IF NOT bGetProgramStateBusy AND intGetProgramStateStep > 0 THEN
	intGetProgramStateStep := 0;
	bRouterBusy := FALSE;
	THIS^.M_LogWarning('M_GetProgramState ended prematurely!');
END_IF
bGetProgramStateBusy := FALSE;

IF NOT bLoadProgramBusy AND intLoadProgramStep > 0 THEN
	intLoadProgramStep := 0;
	bRouterBusy := FALSE;
	THIS^.M_LogWarning('M_LoadProgram ended prematurely!');
END_IF
bLoadProgramBusy := FALSE;

IF NOT bPauseProgramBusy AND intPauseProgramStep > 0 THEN
	intPauseProgramStep := 0;
	bRouterBusy := FALSE;
	THIS^.M_LogWarning('M_PauseProgram ended prematurely!');
END_IF
bPauseProgramBusy := FALSE;

IF NOT bStartProgramBusy AND intStartProgramStep > 0 THEN
	intStartProgramStep := 0;
	bRouterBusy := FALSE;
	THIS^.M_LogWarning('M_StartProgram ended prematurely!');
END_IF
bStartProgramBusy := FALSE;

IF NOT bStopProgramBusy AND intStopProgramStep > 0 THEN
	intStopProgramStep := 0;
	bRouterBusy := FALSE;
	THIS^.M_LogWarning('M_StopProgram ended prematurely!');
END_IF
bStopProgramBusy := FALSE;

IF NOT bResetBusy AND intResetStep > 0 THEN
	intResetStep := 0;
	bRouterBusy := FALSE;
	THIS^.M_LogWarning('M_ResetBusy ended prematurely!');
END_IF
bResetBusy := FALSE;

IF NOT bAbortBusy AND intAbortStep > 0 THEN
	intAbortStep := 0;
	bRouterBusy := FALSE;
	THIS^.M_LogWarning('M_Abort ended prematurely!');
END_IF
bAbortBusy := FALSE;

IF NOT bRouterHelperBusy AND intRouterHelperStep > 0 THEN
	intRouterHelperStep := 0;
	bRouterBusy := FALSE;
	THIS^.M_LogWarning('M_RouterHelper ended prematurely!');
END_IF
bRouterHelperBusy := FALSE;
END_ACTION

(* This method is a template for any methods that use the API. *)
METHOD M_CommandTemplate : BOOL
VAR CONSTANT
	_strCOMMAND_NAME : T_MaxString	:= 'CommandTemplate'; // Name of the API method
	_timeCOMMAND_TIMEOUT : TIME		:= T#30S; // Max time to receive API response
	_strSTART_MSG : T_MaxString		:= 'Routing command...'; // Prints when method starts
	_strEND_MSG : T_MaxString		:= 'Command complete.'; // Prints when method finishes
	_udintERROR_ID : UDINT			:= E_ApiDeviceError.CommandFault; // Error ID to set if command fails
	_strERROR_MSG : T_MaxString		:= 'Command failed!'; // Error message to set if command fails
END_VAR
VAR_INST
	_inst_arrParams: T_ApiParameterList; // Parameters array
	_inst_arrOutputs: T_ApiParameterList; // Outputs array
	_inst_strRet: T_ApiParamValue; // Return string from the router
	_inst_intStep: INT; // Current method step
	_inst_fbParams: FB_ApiParamBuilder; // Parameter builder FB
END_VAR
VAR
	_bComplete: BOOL; // True if the routing finishes
	_intRet: INT; // Return string converted to an integer
	_bResult : BOOL; // Output of the method
	_pArgs: PVOID; // Arguments pointer
END_VAR
_bResult := FALSE;

// Recover from premature stop
(* TEMPLATE: Replace bTemplateBusy and intTemplateStep with relevant
	variables for specific command. Also replace M_CommandTemplate
	and intTemplateStep in the last two lines of this method. *)
bTemplateBusy := TRUE;
_inst_intStep := intTemplateStep;

// Steps
(* TEMPLATE: Parameters should be added in step 10, and output
	parsing should be added in step 30. *)
CASE _inst_intStep OF
	0: // Wait for no error and router not busy
		IF NOT THIS^.P_bError AND NOT bRouterBusy THEN
			bRouterBusy := TRUE;
			_inst_intStep := _inst_intStep + 10;
		END_IF
		
	10: // Initialize parameters
		THIS^.M_LogMessage(_strSTART_MSG);
		_inst_fbParams.M_ClearParameters();
		_pArgs := _inst_fbParams.M_AddEmptyStruct('args');
		// TEMPLATE: Add any parameters here
		_inst_fbParams.M_OutputToParameterList(_inst_arrParams);
		_inst_intStep := _inst_intStep + 10;
		
	20: // Route the command
		_bComplete := M_RouterHelper(
			_in_strMethodName := _strCOMMAND_NAME, 
			_in_timeTimeout := _timeCOMMAND_TIMEOUT,
			_inout_arrParams := _inst_arrParams,
			_inout_arrOutputs := _inst_arrOutputs,
			_out_strReturnValue=>_inst_strRet);
		
		// If route completed, move to next step
		IF _bComplete THEN
			_inst_intStep := _inst_intStep + 10;
			bRouterBusy := FALSE;
		ELSIF THIS^.P_bError THEN
			_inst_intStep := 0;
			bRouterBusy := FALSE;
		END_IF
		
	30: // Parse results
		_intRet := STRING_TO_INT(_inst_strRet);
		IF _intRet > 0 THEN
			_bResult := TRUE;
			THIS^.M_LogMessage(_strEND_MSG);
			_inst_fbParams.M_LoadFromParameterList(_inst_arrOutputs);
			// TEMPLATE: Do any parsing here
			
		// Set error if command failed
		ELSE
			THIS^.M_SetError(_udintERROR_ID, _strERROR_MSG);
		END_IF
		
		// Go back to start
		_inst_intStep := 0;
END_CASE
// TEMPLATE: Replace with method name and step variable
M_CommandTemplate := _bResult;
intTemplateStep := _inst_intStep;
END_METHOD

(*
Sends the given method to the API and receives and partially parses the result.
*)
METHOD PRIVATE M_RouterHelper : BOOL
VAR_INPUT
	(* Name of the method to call. *)
	_in_strMethodName : T_MaxString;
	(* Maximum time to wait for method response. *)
	_in_timeTimeout : TIME;
END_VAR
VAR_IN_OUT
	(* The array of parameters to send to the API. *)
	_inout_arrParams : T_ApiParameterList;
	(* The array that gets populated with any method output data. *)
	_inout_arrOutputs : T_ApiParameterList;
END_VAR
VAR_OUTPUT
	(* JSON string of the method return value. *)
	_out_strReturnValue: T_ApiParamValue;
END_VAR
VAR_INST
	(* Current step. *)
	_inst_intStep: INT;
	(* True if the method executed. *)
	_inst_bExec: BOOL;
	(* Return string of the method. *)
	_inst_strRet: T_ApiParamValue;
END_VAR
VAR
	(* True once the command routing finishes. *)
	_bComplete: BOOL;
	(* True once the API connects. *)
	_bApiConnect: BOOL;
END_VAR
// Recover from premature stop
bRouterHelperBusy := TRUE;
_inst_intStep := intRouterHelperStep;

// Steps
CASE _inst_intStep OF
	0: // Start process only if there is no error on this FB
		IF NOT THIS^.P_bError THEN
			in_fbApi.M_ClearError();
			_inst_intStep := 10;
		END_IF
		
	10: // Check if command router is connected
		IF NOT in_fbApi.P_bConnected THEN
			_inst_intStep := 20; // Go to API connect step
		ELSE
			_inst_intStep := 30; // Go to route command step
		END_IF
		
	20: // Connect to the command router
		_bApiConnect := in_fbApi.M_Connect();
		IF _bApiConnect THEN
			_inst_intStep := _inst_intStep + 10; // Go to next step
		ELSIF in_fbApi.P_bError THEN
			THIS^.M_SetError(E_ApiDeviceError.CommandRouterError, 'Error on command router function block while connecting!');
			_inst_intStep := 0; // Go back to start
		END_IF
		
	30:	// Route the command
		_bComplete := in_fbApi.M_RouteCommand(
			_in_strModuleId := in_strApiModuleId,
			_in_strMethodName := _in_strMethodName,
			_in_timeTimeout := _in_timeTimeout,
			_inout_arrParameters := _inout_arrParams,
			_inout_arrOutputs := _inout_arrOutputs,
			_out_bCommandExecuted => _inst_bExec,
			_out_strReturnValue => _inst_strRet);
		IF _bComplete THEN
			_inst_intStep := _inst_intStep + 10; // Go to next step
		ELSIF in_fbApi.P_bError THEN
			THIS^.M_SetError(E_ApiDeviceError.CommandRouterError, 'Error on command router function block while routing command!');
			_inst_intStep := 0; // Go back to start
		END_IF
		
	40: // Check result then go back to start
		IF NOT _inst_bExec THEN
			THIS^.M_SetError(E_ApiDeviceError.CommandFault, 'Method in API failed to execute!');
		ELSE
			_out_strReturnValue := _inst_strRet;
			M_RouterHelper := TRUE;
		END_IF
		_inst_intStep := 0; // Go back to start
END_CASE

intRouterHelperStep := _inst_intStep;
END_METHOD

END_FUNCTION_BLOCK

// Concrete/API/FB_ApiParamBuilder
(*
Used to build an array of correctly-formatted ST_ApiParameter structs.

Use M_AddParameter to add a parameter to the parameters list.

If a parameter is a struct or array, use M_AddStructMember and M_AddArrayElement
respectively after M_AddParameter to manually build the struct or array in this
function block.

Use M_ClearParameters to clear the memory, and M_GetParameterList to get
the correctly formatted T_ApiParameters object.
*)
FUNCTION_BLOCK FB_ApiParamBuilder EXTENDS FB_Module
VAR_INPUT
END_VAR
VAR_OUTPUT
END_VAR
VAR
	fbJson : FB_JsonDynDomParser;
	pJsonDoc: Tc3_JsonXml.PVOID;
	bInitialized: BOOL := FALSE;
END_VAR

(* Appends a new element to the array given by the pointer and returns a
	pointer to the added value. Supports most primitive types directly.

	If the value is an array, will only add a blank array that must be populated
	manually by calling M_AddArrayElement with the pointer returned by this method. 

	If the value is a struct, will only add a blank struct that must be populated
	manually by calling M_AddStructMember with the pointer returned by this method. 

	Value will be stored as null if the value type is not yet supported. *)
METHOD M_AddArrayElement : PVOID
VAR_INPUT
	(* Pointer to the array that should be added to. This pointer is returned
		by any M_Add<item> methods that were used to add an array. *)
	_in_pArrayPointer : PVOID;
	
	(* The value to append to the array. *)
	_in_anyValue : ANY;
END_VAR
IF NOT bInitialized THEN
	RETURN;
ELSIF NOT fbJson.IsArray(_in_pArrayPointer) THEN
	RETURN;
END_IF

M_AddArrayElement := M_Pushback(_in_pArrayPointer, _in_anyValue);
END_METHOD

(* Adds a new empty array parameter. Use M_AddArrayElement with
	the output PVOID of this to populate. *)
METHOD M_AddEmptyArray : PVOID
VAR_INPUT
	(* Parameter name. *)
	_in_strKey : T_MaxString;
END_VAR
VAR
	_arrRef: ARRAY[1..2] OF BOOL;
END_VAR
IF NOT bInitialized THEN
	pJsonDoc := fbJson.NewDocument();
	bInitialized := TRUE;
END_IF

M_AddEmptyArray := THIS^.M_Add(pJsonDoc, _in_strKey, _arrRef);
END_METHOD

(* Appends a new empty array to the array given by the pointer and returns a
	pointer to the added array.*)
METHOD M_AddEmptyArrayToArray : PVOID
VAR_INPUT
	(* Pointer to the array that should be added to. This pointer is returned
		by any M_Add<item> methods that were used to add an array. *)
	_in_pArrayPointer : PVOID;
END_VAR
VAR
	_arrRef: ARRAY[1..2] OF BOOL;
END_VAR
IF NOT bInitialized THEN
	M_AddEmptyArrayToArray := 0;
	RETURN;
ELSIF NOT fbJson.IsArray(_in_pArrayPointer) THEN
	M_AddEmptyArrayToArray := 0;
	RETURN;
END_IF

M_AddEmptyArrayToArray := M_Pushback(_in_pArrayPointer, _arrRef);
END_METHOD

(* Adds a new empty struct with the given key to the given struct pointer and 
	returns a pointer to the added value.*)
METHOD M_AddEmptyArrayToStruct : PVOID
VAR_INPUT
	(* Pointer to the struct that should be added to. This pointer is returned
		by any M_Add<item> methods that were used to add a struct. *)
	_in_pStructPointer : PVOID;
	
	(* Key to add to the struct. *)
	_in_strKey : T_MaxString;
END_VAR
VAR
	_arrRef: ARRAY[1..2] OF BOOL;
END_VAR
IF NOT bInitialized THEN
	M_AddEmptyArrayToStruct := 0;
	RETURN;
ELSIF NOT fbJson.IsObject(_in_pStructPointer) THEN
	M_AddEmptyArrayToStruct := 0;
	RETURN;
END_IF

M_AddEmptyArrayToStruct := M_Add(_in_pStructPointer, _in_strKey, _arrRef);
END_METHOD

(* Adds a new empty struct with the given parameter name. Use M_AddStructMember
	with the PVOID output of this to populate. *)
METHOD M_AddEmptyStruct : PVOID
VAR_INPUT
	(* Parameter name. *)
	_in_strKey : T_MaxString;
END_VAR
VAR
	_stRef: ST_ApiParameter;
END_VAR
IF NOT bInitialized THEN
	pJsonDoc := fbJson.NewDocument();
	bInitialized := TRUE;
END_IF

M_AddEmptyStruct := THIS^.M_Add(pJsonDoc, _in_strKey, _stRef);
END_METHOD

(* Appends a new empty struct to the array given by the pointer and returns a
	pointer to the added struct. *)
METHOD M_AddEmptyStructToArray : PVOID
VAR_INPUT
	(* Pointer to the array that should be added to. This pointer is returned
		by any M_Add<item> methods that were used to add an array. *)
	_in_pArrayPointer : PVOID;
END_VAR
VAR
	_stRef: ST_ApiParameter;
END_VAR
IF NOT bInitialized THEN
	M_AddEmptyStructToArray := 0;
	RETURN;
ELSIF NOT fbJson.IsArray(_in_pArrayPointer) THEN
	M_AddEmptyStructToArray := 0;
	RETURN;
END_IF

M_AddEmptyStructToArray := M_Pushback(_in_pArrayPointer, _stRef);
END_METHOD

(* Adds a new empty struct with the given key to the given struct pointer and 
	returns a pointer to the added value.*)
METHOD M_AddEmptyStructToStruct : PVOID
VAR_INPUT
	(* Pointer to the struct that should be added to. This pointer is returned
		by any M_Add<item> methods that were used to add a struct. *)
	_in_pStructPointer : PVOID;
	
	(* Key to add to the struct. *)
	_in_strKey : T_MaxString;
END_VAR
VAR
	_stRef: ST_ApiParameter;
END_VAR
IF NOT bInitialized THEN
	M_AddEmptyStructToStruct := 0;
	RETURN;
ELSIF NOT fbJson.IsObject(_in_pStructPointer) THEN
	M_AddEmptyStructToStruct := 0;
	RETURN;
END_IF

M_AddEmptyStructToStruct := M_Add(_in_pStructPointer, _in_strKey, _stRef);
END_METHOD

(* Adds a new key:value pair to the parameters list and returns a pointer to
	the added value. Supports most primitive types directly.

	If the value is an array, will only add a blank array that must be populated
	manually by calling M_AddArrayElement with the pointer returned by this method. 

	If the value is a struct, will only add a blank struct that must be populated
	manually by calling M_AddStructMember with the pointer returned by this method. 

	Value will be stored as null if the value type is not yet supported. *)
METHOD M_AddParameter : PVOID
VAR_INPUT
	(* Parameter name. *)
	_in_strKey : T_MaxString;
	
	(* Parameter value. *)
	_in_anyValue : ANY;
END_VAR
VAR
	_pJsonMember: Tc3_JsonXml.PVOID;
END_VAR
IF NOT bInitialized THEN
	pJsonDoc := fbJson.NewDocument();
	bInitialized := TRUE;
END_IF

_pJsonMember := THIS^.M_Add(pJsonDoc, _in_strKey, _in_anyValue);

M_AddParameter := _pJsonMember;
END_METHOD

(* Adds a new key:value pair to the parameters list and returns a pointer to
	the added value. Supports most primitive types directly.

	If the value is an array, will only add a blank array that must be populated
	manually by calling M_AddArrayElement with the pointer returned by this method. 

	If the value is a struct, will only add a blank struct that must be populated
	manually by calling M_AddStructMember with the pointer returned by this method. 

	Value will be stored as null if the value type is not yet supported. *)
METHOD M_AddStructMember : PVOID
VAR_INPUT
	(* Pointer to the struct that should be added to. This pointer is returned
		by any M_Add<item> methods that were used to add a struct. *)
	_in_pStructPointer : PVOID;
	
	(* Key to add to the struct. *)
	_in_strKey : T_MaxString;
	
	(* Value to add to the struct. *)
	_in_anyValue : ANY;
END_VAR
IF NOT bInitialized THEN
	M_AddStructMember := 0;
	RETURN;
ELSIF NOT fbJson.IsObject(_in_pStructPointer) THEN
	M_AddStructMember := 0;
	RETURN;
END_IF

M_AddStructMember := M_Add(_in_pStructPointer, _in_strKey, _in_anyValue);
END_METHOD

(* Clears all current parameters. *)
METHOD M_ClearParameters : BOOL
VAR_INPUT
END_VAR
VAR
END_VAR
pJsonDoc := fbJson.NewDocument();
bInitialized := TRUE;
END_METHOD

(* Populates the given parameters list with the added key:value pairs. *)
METHOD M_OutputToParameterList : BOOL
VAR_INPUT
END_VAR
VAR_IN_OUT
	// Parameters list to populate.
	_inout_arrParameters : T_ApiParameterList;
END_VAR
VAR
	_dintParamMin: DINT; // Lower bound of parameters array
	_dintParamMax: DINT; // Upper bound of parameters array
	_dintParamIndex: DINT; // Current parameters array index
	_pJsonIterator: Tc3_JsonXml.PVOID; // Current JSON iterator pointer
	_pJsonIteratorEnd: Tc3_JsonXml.PVOID; // JSON iterator end pointer
	_strName: STRING; // Name of the parameter
	_pValue: Tc3_JsonXml.PVOID; // Pointer to the parameter
	_strValue: T_ApiParamValue; // Parameter value
END_VAR
// Get the array bounds
_dintParamMin := GVL_Api.dintPARAM_LOWER_BOUND;
_dintParamMax := GVL_Api.dintPARAM_UPPER_BOUND;

// Clear the array
FOR _dintParamIndex := _dintParamMin TO _dintParamMax DO
	_inout_arrParameters[_dintParamIndex].strKey := '';
	_inout_arrParameters[_dintParamIndex].strValue := '';
END_FOR

// Initialize the iterators
_dintParamIndex := _dintParamMin;
_pJsonIterator := fbJson.MemberBegin(pJsonDoc);
_pJsonIteratorEnd := fbJson.MemberEnd(pJsonDoc);

// Populate each array member. If there are more parameters than there are
// array members, will stop iterating.
WHILE _pJsonIterator <> _pJsonIteratorEnd AND _dintParamIndex <= _dintParamMax DO
	_strName := fbJson.GetMemberName(_pJsonIterator);
	_pValue := fbJson.GetMemberValue(_pJsonIterator);
	MEMSET(ADR(_strValue),0,SIZEOF(_strValue));
	fbJson.CopyJson(_pValue, _strValue, SIZEOF(_strValue));
	_inout_arrParameters[_dintParamIndex].strKey := _strName;
	_inout_arrParameters[_dintParamIndex].strValue := _strValue;
	_pJsonIterator := fbJson.NextMember(_pJsonIterator);
	_dintParamIndex := _dintParamIndex + 1;
END_WHILE

M_OutputToParameterList := TRUE;
END_METHOD

(* Adds a key:value pair to the given struct. *)
METHOD PRIVATE M_Add : PVOID
VAR_INPUT
	_in_pJsonPointer : PVOID;
	_in_strKey : T_MaxString;
	_in_anyValue : ANY;
END_VAR
VAR
	_pJsonMember: Tc3_JsonXml.PVOID; // Pointer to the added JSON member

	// Supported types
	_pBoolValue:		POINTER TO BOOL;
	_pInt32Value:		POINTER TO DINT;
	_pUint32Value:		POINTER TO UINT;
	_pInt64Value:		POINTER TO LINT;
	_pUint64Value:		POINTER TO ULINT;
	_pDoubleValue:		POINTER TO LREAL;
	_pDateTimeValue:	POINTER TO DATE_AND_TIME;
	_pStringValue:		POINTER TO STRING;
	
	// Converted types
	_pSingleValue:		POINTER TO REAL;
	_pInt16Value:		POINTER TO INT;
	_pInt8Value:		POINTER TO SINT;
	_pUint16Value:		POINTER TO UINT;
	_pUint8Value:		POINTER TO USINT;
	_pByteValue:		POINTER TO BYTE;
	_pWordValue:		POINTER TO WORD;
	_pDwordValue:		POINTER TO DWORD;
	_pLwordValue:		POINTER TO LWORD;
	_pDateValue:		POINTER TO DATE;
	_pTimeValue:		POINTER TO TIME;
	
	// Converted type values
	_lrealSingleValue:	LREAL;
	_dintInt16Value:	DINT;
	_dintInt8Value:		DINT;
	_udintUint16Value:	UDINT;
	_udintUint8Value:	UDINT;
	_udintByteValue:	UDINT;
	_udintWordValue:	UDINT;
	_udintDwordValue:	UDINT;
	_ulintLwordValue:	ULINT;
	_dtDateValue:		DATE_AND_TIME;
	_dtTimeValue:		DATE_AND_TIME;
END_VAR
// Add key-value pair to JSON doc based on type
CASE _in_anyValue.TypeClass OF
	// Supported datatypes
	__SYSTEM.TYPE_CLASS.TYPE_BOOL:
		_pBoolValue := _in_anyValue.pValue;
		_pJsonMember := fbJson.AddBoolMember(_in_pJsonPointer, _in_strKey, _pBoolValue^);
	__SYSTEM.TYPE_CLASS.TYPE_DATEANDTIME:
		_pDateTimeValue := _in_anyValue.pValue;
		_pJsonMember := fbJson.AddDateTimeMember(_in_pJsonPointer, _in_strKey, _pDateTimeValue^);
	__SYSTEM.TYPE_CLASS.TYPE_LREAL:
		_pDoubleValue := _in_anyValue.pValue;
		_pJsonMember := fbJson.AddDoubleMember(_in_pJsonPointer, _in_strKey, _pDoubleValue^);
	__SYSTEM.TYPE_CLASS.TYPE_LINT:
		_pInt64Value := _in_anyValue.pValue;
		_pJsonMember := fbJson.AddInt64Member(_in_pJsonPointer, _in_strKey, _pInt64Value^);
	__SYSTEM.TYPE_CLASS.TYPE_DINT:
		_pInt32Value := _in_anyValue.pValue;
		_pJsonMember := fbJson.AddIntMember(_in_pJsonPointer, _in_strKey, _pInt32Value^);
	__SYSTEM.TYPE_CLASS.TYPE_STRING:
		_pStringValue := _in_anyValue.pValue;
		_pJsonMember := fbJson.AddStringMember(_in_pJsonPointer, _in_strKey, _pStringValue^);
	__SYSTEM.TYPE_CLASS.TYPE_ULINT:
		_pUint64Value := _in_anyValue.pValue;
		_pJsonMember := fbJson.AddUint64Member(_in_pJsonPointer, _in_strKey, _pUint64Value^);
	__SYSTEM.TYPE_CLASS.TYPE_UDINT:
		_pUint32Value := _in_anyValue.pValue;
		_pJsonMember := fbJson.AddUintMember(_in_pJsonPointer, _in_strKey, _pUint32Value^);
		
	// Converted datatypes
	__SYSTEM.TYPE_CLASS.TYPE_REAL:
		_pSingleValue := _in_anyValue.pValue;
		_lrealSingleValue := REAL_TO_LREAL(_pSingleValue^);
		_pJsonMember := fbJson.AddDoubleMember(_in_pJsonPointer, _in_strKey, _lrealSingleValue);
	__SYSTEM.TYPE_CLASS.TYPE_INT:
		_pInt16Value := _in_anyValue.pValue;
		_dintInt16Value := INT_TO_DINT(_pInt16Value^);
		_pJsonMember := fbJson.AddIntMember(_in_pJsonPointer, _in_strKey, _dintInt16Value);
	__SYSTEM.TYPE_CLASS.TYPE_SINT:
		_pInt8Value := _in_anyValue.pValue;
		_dintInt8Value := SINT_TO_DINT(_pInt8Value^);
		_pJsonMember := fbJson.AddIntMember(_in_pJsonPointer, _in_strKey, _dintInt8Value);
	__SYSTEM.TYPE_CLASS.TYPE_UINT:
		_pUint16Value := _in_anyValue.pValue;
		_udintUint16Value := UINT_TO_UDINT(_pUint16Value^);
		_pJsonMember := fbJson.AddUintMember(_in_pJsonPointer, _in_strKey, _udintUint16Value);
	__SYSTEM.TYPE_CLASS.TYPE_USINT:
		_pUint8Value := _in_anyValue.pValue;
		_udintUint8Value := USINT_TO_UDINT(_pUint8Value^);
		_pJsonMember := fbJson.AddUintMember(_in_pJsonPointer, _in_strKey, _udintUint8Value);
	__SYSTEM.TYPE_CLASS.TYPE_BYTE:
		_pByteValue := _in_anyValue.pValue;
		_udintByteValue := BYTE_TO_UDINT(_pByteValue^);
		_pJsonMember := fbJson.AddUintMember(_in_pJsonPointer, _in_strKey, _udintByteValue);
	__SYSTEM.TYPE_CLASS.TYPE_WORD:
		_pWordValue := _in_anyValue.pValue;
		_udintWordValue := WORD_TO_UDINT(_pWordValue^);
		_pJsonMember := fbJson.AddUintMember(_in_pJsonPointer, _in_strKey, _udintWordValue);
	__SYSTEM.TYPE_CLASS.TYPE_DWORD:
		_pDwordValue := _in_anyValue.pValue;
		_udintDwordValue := DWORD_TO_UDINT(_pDwordValue^);
		_pJsonMember := fbJson.AddUintMember(_in_pJsonPointer, _in_strKey, _udintDwordValue);
	__SYSTEM.TYPE_CLASS.TYPE_LWORD:
		_pLwordValue := _in_anyValue.pValue;
		_ulintLwordValue := LWORD_TO_ULINT(_pLwordValue^);
		_pJsonMember := fbJson.AddUint64Member(_in_pJsonPointer, _in_strKey, _ulintLwordValue);
	__SYSTEM.TYPE_CLASS.TYPE_DATE:
		_pDateValue := _in_anyValue.pValue;
		_dtDateValue := DATE_TO_DT(_pDateValue^);
		_pJsonMember := fbJson.AddDateTimeMember(_in_pJsonPointer, _in_strKey, _dtDateValue);
	__SYSTEM.TYPE_CLASS.TYPE_TIME:
		_pTimeValue := _in_anyValue.pValue;
		_dtTimeValue := TIME_TO_DT(_pTimeValue^);
		_pJsonMember := fbJson.AddDateTimeMember(_in_pJsonPointer, _in_strKey, _dtTimeValue);
		
	// Empty objects
	__SYSTEM.TYPE_CLASS.TYPE_ARRAY:
		_pJsonMember := fbJson.AddArrayMember(_in_pJsonPointer, _in_strKey, 0);
	__SYSTEM.TYPE_CLASS.TYPE_USERDEF:
		_pJsonMember := fbJson.AddObjectMember(_in_pJsonPointer, _in_strKey);
		
ELSE
	_pJsonMember := fbJson.AddNullMember(_in_pJsonPointer,_in_strKey);
END_CASE

M_Add := _pJsonMember;
END_METHOD

(* Adds an element to the given array. *)
METHOD PRIVATE M_Pushback : PVOID
VAR_INPUT
	_in_pJsonPointer : PVOID;
	_in_anyValue : ANY;
END_VAR
VAR
	_pJsonMember: Tc3_JsonXml.PVOID;  // Pointer to the added JSON member

	// Supported types
	_pBoolValue:		POINTER TO BOOL;
	_pInt32Value:		POINTER TO DINT;
	_pUint32Value:		POINTER TO UINT;
	_pInt64Value:		POINTER TO LINT;
	_pUint64Value:		POINTER TO ULINT;
	_pDoubleValue:		POINTER TO LREAL;
	_pDateTimeValue:	POINTER TO DATE_AND_TIME;
	_pStringValue:		POINTER TO STRING;
	
	// Converted types
	_pSingleValue:		POINTER TO REAL;
	_pInt16Value:		POINTER TO INT;
	_pInt8Value:		POINTER TO SINT;
	_pUint16Value:		POINTER TO UINT;
	_pUint8Value:		POINTER TO USINT;
	_pByteValue:		POINTER TO BYTE;
	_pWordValue:		POINTER TO WORD;
	_pDwordValue:		POINTER TO DWORD;
	_pLwordValue:		POINTER TO LWORD;
	_pDateValue:		POINTER TO DATE;
	_pTimeValue:		POINTER TO TIME;
	
	// Converted type values
	_lrealSingleValue:	LREAL;
	_dintInt16Value:	DINT;
	_dintInt8Value:		DINT;
	_udintUint16Value:	UDINT;
	_udintUint8Value:	UDINT;
	_udintByteValue:	UDINT;
	_udintWordValue:	UDINT;
	_udintDwordValue:	UDINT;
	_ulintLwordValue:	ULINT;
	_dtDateValue:		DATE_AND_TIME;
	_dtTimeValue:		DATE_AND_TIME;
END_VAR
// Add key-value pair to JSON doc based on type
CASE _in_anyValue.TypeClass OF
	// Supported
	__SYSTEM.TYPE_CLASS.TYPE_BOOL:
		_pBoolValue := _in_anyValue.pValue;
		_pJsonMember := fbJson.PushbackBoolValue(_in_pJsonPointer, _pBoolValue^);
	__SYSTEM.TYPE_CLASS.TYPE_DATEANDTIME:
		_pDateTimeValue := _in_anyValue.pValue;
		_pJsonMember := fbJson.PushbackDateTimeValue(_in_pJsonPointer, _pDateTimeValue^);
	__SYSTEM.TYPE_CLASS.TYPE_LREAL:
		_pDoubleValue := _in_anyValue.pValue;
		_pJsonMember := fbJson.PushbackDoubleValue(_in_pJsonPointer, _pDoubleValue^);
	__SYSTEM.TYPE_CLASS.TYPE_LINT:
		_pInt64Value := _in_anyValue.pValue;
		_pJsonMember := fbJson.PushbackInt64Value(_in_pJsonPointer, _pInt64Value^);
	__SYSTEM.TYPE_CLASS.TYPE_DINT:
		_pInt32Value := _in_anyValue.pValue;
		_pJsonMember := fbJson.PushbackIntValue(_in_pJsonPointer, _pInt32Value^);
	__SYSTEM.TYPE_CLASS.TYPE_STRING:
		_pStringValue := _in_anyValue.pValue;
		_pJsonMember := fbJson.PushbackStringValue(_in_pJsonPointer, _pStringValue^);
	__SYSTEM.TYPE_CLASS.TYPE_ULINT:
		_pUint64Value := _in_anyValue.pValue;
		_pJsonMember := fbJson.PushbackUint64Value(_in_pJsonPointer, _pUint64Value^);
	__SYSTEM.TYPE_CLASS.TYPE_UDINT:
		_pUint32Value := _in_anyValue.pValue;
		_pJsonMember := fbJson.PushbackUintValue(_in_pJsonPointer, _pUint32Value^);
		
	// Converted
	__SYSTEM.TYPE_CLASS.TYPE_REAL:
		_pSingleValue := _in_anyValue.pValue;
		_lrealSingleValue := REAL_TO_LREAL(_pSingleValue^);
		_pJsonMember := fbJson.PushbackDoubleValue(_in_pJsonPointer, _lrealSingleValue);
	__SYSTEM.TYPE_CLASS.TYPE_INT:
		_pInt16Value := _in_anyValue.pValue;
		_dintInt16Value := INT_TO_DINT(_pInt16Value^);
		_pJsonMember := fbJson.PushbackIntValue(_in_pJsonPointer, _dintInt16Value);
	__SYSTEM.TYPE_CLASS.TYPE_SINT:
		_pInt8Value := _in_anyValue.pValue;
		_dintInt8Value := SINT_TO_DINT(_pInt8Value^);
		_pJsonMember := fbJson.PushbackIntValue(_in_pJsonPointer, _dintInt8Value);
	__SYSTEM.TYPE_CLASS.TYPE_UINT:
		_pUint16Value := _in_anyValue.pValue;
		_udintUint16Value := UINT_TO_UDINT(_pUint16Value^);
		_pJsonMember := fbJson.PushbackUintValue(_in_pJsonPointer, _udintUint16Value);
	__SYSTEM.TYPE_CLASS.TYPE_USINT:
		_pUint8Value := _in_anyValue.pValue;
		_udintUint8Value := USINT_TO_UDINT(_pUint8Value^);
		_pJsonMember := fbJson.PushbackUintValue(_in_pJsonPointer, _udintUint8Value);
	__SYSTEM.TYPE_CLASS.TYPE_BYTE:
		_pByteValue := _in_anyValue.pValue;
		_udintByteValue := BYTE_TO_UDINT(_pByteValue^);
		_pJsonMember := fbJson.PushbackUintValue(_in_pJsonPointer, _udintByteValue);
	__SYSTEM.TYPE_CLASS.TYPE_WORD:
		_pWordValue := _in_anyValue.pValue;
		_udintWordValue := WORD_TO_UDINT(_pWordValue^);
		_pJsonMember := fbJson.PushbackUintValue(_in_pJsonPointer, _udintWordValue);
	__SYSTEM.TYPE_CLASS.TYPE_DWORD:
		_pDwordValue := _in_anyValue.pValue;
		_udintDwordValue := DWORD_TO_UDINT(_pDwordValue^);
		_pJsonMember := fbJson.PushbackUintValue(_in_pJsonPointer, _udintDwordValue);
	__SYSTEM.TYPE_CLASS.TYPE_LWORD:
		_pLwordValue := _in_anyValue.pValue;
		_ulintLwordValue := LWORD_TO_ULINT(_pLwordValue^);
		_pJsonMember := fbJson.PushbackUint64Value(_in_pJsonPointer, _ulintLwordValue);
	__SYSTEM.TYPE_CLASS.TYPE_DATE:
		_pDateValue := _in_anyValue.pValue;
		_dtDateValue := DATE_TO_DT(_pDateValue^);
		_pJsonMember := fbJson.PushbackDateTimeValue(_in_pJsonPointer, _dtDateValue);
	__SYSTEM.TYPE_CLASS.TYPE_TIME:
		_pTimeValue := _in_anyValue.pValue;
		_dtTimeValue := TIME_TO_DT(_pTimeValue^);
		_pJsonMember := fbJson.PushbackDateTimeValue(_in_pJsonPointer, _dtTimeValue);
	
	// Objects
	__SYSTEM.TYPE_CLASS.TYPE_ARRAY:
		_pJsonMember := fbJson.PushbackJsonValue(_in_pJsonPointer, '[]');
	__SYSTEM.TYPE_CLASS.TYPE_USERDEF:
		_pJsonMember := fbJson.PushbackJsonValue(_in_pJsonPointer, '{}');
ELSE
	_pJsonMember := fbJson.PushbackNullValue(_in_pJsonPointer);
END_CASE

M_Pushback := _pJsonMember;
END_METHOD

METHOD M_ParseBool : BOOL
VAR_INPUT
	(* Pointer to the value. *)
	_in_pValuePointer : PVOID;
END_VAR
IF _in_pValuePointer = 0 THEN
	THIS^.M_LogWarning('Invalid pointer in M_ParseBool!');
	RETURN;
END_IF
IF fbJson.IsBool(_in_pValuePointer) THEN
	M_ParseBool := fbJson.GetBool(_in_pValuePointer);
END_IF
END_METHOD

METHOD M_ParseDateTime : DATE_AND_TIME
VAR_INPUT
	(* Pointer to the value. *)
	_in_pValuePointer : PVOID;
END_VAR
IF _in_pValuePointer = 0 THEN
	THIS^.M_LogWarning('Invalid pointer in M_ParseDateTime!');
	RETURN;
END_IF
IF fbJson.IsISO8601TimeFormat(_in_pValuePointer) THEN
	M_ParseDateTime := fbJson.GetDateTime(_in_pValuePointer);
END_IF
END_METHOD

METHOD M_ParseDouble : LREAL
VAR_INPUT
	(* Pointer to the value. *)
	_in_pValuePointer : PVOID;
END_VAR
IF _in_pValuePointer = 0 THEN
	THIS^.M_LogWarning('Invalid pointer in M_ParseDouble!');
	RETURN;
END_IF
IF fbJson.IsDouble(_in_pValuePointer) THEN
	M_ParseDouble := fbJson.GetDouble(_in_pValuePointer);
END_IF
END_METHOD

METHOD M_ParseInt : DINT
VAR_INPUT
	(* Pointer to the value. *)
	_in_pValuePointer : PVOID;
END_VAR
IF _in_pValuePointer = 0 THEN
	THIS^.M_LogWarning('Invalid pointer in M_ParseInt!');
	RETURN;
END_IF
IF fbJson.IsInt(_in_pValuePointer) THEN
	M_ParseInt := fbJson.GetInt(_in_pValuePointer);
END_IF
END_METHOD

METHOD M_ParseInt64 : LINT
VAR_INPUT
	(* Pointer to the value. *)
	_in_pValuePointer : PVOID;
END_VAR
IF _in_pValuePointer = 0 THEN
	THIS^.M_LogWarning('Invalid pointer in M_ParseInt64!');
	RETURN;
END_IF
IF fbJson.IsInt64(_in_pValuePointer) THEN
	M_ParseInt64 := fbJson.GetInt64(_in_pValuePointer);
END_IF
END_METHOD

METHOD M_ParseString : T_MaxString
VAR_INPUT
	(* Pointer to the value. *)
	_in_pValuePointer : PVOID;
END_VAR
IF _in_pValuePointer = 0 THEN
	THIS^.M_LogWarning('Invalid pointer in M_ParseString!');
	RETURN;
END_IF
IF fbJson.IsString(_in_pValuePointer) THEN
	M_ParseString := fbJson.GetString(_in_pValuePointer);
END_IF
END_METHOD

METHOD M_ParseUint : UDINT
VAR_INPUT
	(* Pointer to the value. *)
	_in_pValuePointer : PVOID;
END_VAR
IF _in_pValuePointer = 0 THEN
	THIS^.M_LogWarning('Invalid pointer in M_ParseUint!');
	RETURN;
END_IF
IF fbJson.IsUint(_in_pValuePointer) THEN
	M_ParseUInt := fbJson.GetUint(_in_pValuePointer);
END_IF
END_METHOD

METHOD M_ParseUint64 : ULINT
VAR_INPUT
	(* Pointer to the value. *)
	_in_pValuePointer : PVOID;
END_VAR
IF _in_pValuePointer = 0 THEN
	THIS^.M_LogWarning('Invalid pointer in M_ParseUint64!');
	RETURN;
END_IF
IF fbJson.IsUint64(_in_pValuePointer) THEN
	M_ParseUInt64 := fbJson.GetUint64(_in_pValuePointer);
END_IF
END_METHOD

(* Returns a pointer to the value of the given array index inside of the
	array given by the pointer. Use the relevant M_Parse<type> method
	to get the data from the value. *)
METHOD M_GetArrayElement : PVOID
VAR_INPUT
	(* Pointer to the struct to get the member from. *)
	_in_pArrayPointer : PVOID;
	(* Index of the element to get. *)
	_in_udintIndex : UDINT;
END_VAR
IF bInitialized THEN
	M_GetArrayElement := fbJson.GetArrayValueByIdx(_in_pArrayPointer, _in_udintIndex);
END_IF
END_METHOD

(* Returns a pointer to the value of the requested parameter. Use the relevant
	M_Parse<type> method to get the data from the value, or M_GetStructMember
	or M_GetArrayElement if the value is a struct or array respectively. *)
METHOD M_GetParameter : PVOID
VAR_INPUT
	(* Name of the parameter to get. *)
	_in_strName : T_MaxString;
END_VAR
M_GetParameter := M_GetStructMember(pJsonDoc, _in_strName);
END_METHOD

(* Returns a pointer to the value of the given parameter inside of the
	struct given by the pointer. Use the relevant M_Parse<type> method
	to get the data from the value. *)
METHOD M_GetStructMember : PVOID
VAR_INPUT
	(* Pointer to the struct to get the member from. *)
	_in_pStructPointer : PVOID;
	(* Name of the parameter to get. *)
	_in_strName : T_MaxString;
END_VAR
IF bInitialized THEN
	M_GetStructMember := fbJson.FindMember(_in_pStructPointer, _in_strName);
END_IF
END_METHOD

METHOD M_LoadFromParameterList : BOOL
VAR_INPUT
END_VAR
VAR_IN_OUT
	// Parameters list to load into the function block.
	_inout_arrParameters : T_ApiParameterList;
END_VAR
VAR
	_dintParamMin: DINT; // Lower bound of the parameters array
	_dintParamMax: DINT; // Upper bound of the parameters array
	_dintParamIndex: DINT; // Current index of the parameters array
	_strKey: STRING(255); // Name of the parameter
	_strValue: T_ApiParamValue; // Value of the parameter
END_VAR
// Clear the JSON doc
pJsonDoc := fbJson.NewDocument();
bInitialized := TRUE;

// Get the array bounds
_dintParamMin := GVL_Api.dintPARAM_LOWER_BOUND;
_dintParamMax := GVL_Api.dintPARAM_UPPER_BOUND;

// Populate the JSON document
FOR _dintParamIndex := _dintParamMin TO _dintParamMax DO
	_strKey := _inout_arrParameters[_dintParamIndex].strKey;
	_strValue := _inout_arrParameters[_dintParamIndex].strValue;
	IF LEN(_strKey) > 0 THEN
		fbJson.AddJsonMember(pJsonDoc, _strKey, _strValue);
	END_IF
END_FOR

M_LoadFromParameterList := TRUE;
END_METHOD

END_FUNCTION_BLOCK

// Concrete/IO Mapping/Obsolete/F_LinkDigitalIOStructs
FUNCTION F_LinkDigitalIOStructs : BOOL
VAR_INPUT
END_VAR
VAR_IN_OUT
	(* The force and force value bits of this will be set to the values of the other. *)
	inout_stControl: ST_DebugDigitalIO;
	(* All info bits of this will be assigned to the control. *)
	inout_stStatus: ST_DebugDigitalIO;
END_VAR
VAR
END_VAR

inout_stStatus.bForce := inout_stControl.bForce;
inout_stStatus.bForceValue := inout_stControl.bForceValue;
inout_stControl.bCurrentValue := inout_stStatus.bCurrentValue;
inout_stControl.strLabel := inout_stStatus.strLabel;

END_FUNCTION

// Concrete/IO Mapping/Obsolete/F_SetDigitalInput
FUNCTION F_SetDigitalInput : BOOL
VAR_INPUT
	in_bValue: BOOL;
	in_strLabel: T_MaxString;
END_VAR
VAR_IN_OUT
	inout_stInput: ST_DebugDigitalIO;
END_VAR
VAR
END_VAR

inout_stInput.bOutput := FALSE;
inout_stInput.bCurrentValue := in_bValue;
inout_stInput.strLabel := in_strLabel;

END_FUNCTION

// Concrete/IO Mapping/Obsolete/F_SetDigitalOutput
FUNCTION F_SetDigitalOutput : BOOL
VAR_INPUT
	in_bValue: BOOL;
	in_strLabel: T_MaxString;
END_VAR
VAR_IN_OUT
	inout_stOutput: ST_DebugDigitalIO;
END_VAR
VAR_OUTPUT
	out_bValue: BOOL;
END_VAR
VAR
END_VAR

inout_stOutput.bOutput := TRUE;
inout_stOutput.strLabel := in_strLabel;
IF inout_stOutput.bForce THEN
	out_bValue := inout_stOutput.bForceValue;
ELSE
	out_bValue := in_bValue;
END_IF
inout_stOutput.bCurrentValue := out_bValue;

END_FUNCTION

// Concrete/IO Mapping/F_LinkDigitalIO
(* Links together to digital IO structs. *)
FUNCTION F_LinkDigitalIO : BOOL
VAR_INPUT
END_VAR
VAR_IN_OUT
	(* The force and force value bits of this will be set to the values of the other. *)
	inout_stControl: ST_DigitalIO;
	(* All info bits of this will be assigned to the control. *)
	inout_stStatus: ST_DigitalIO;
END_VAR
VAR
END_VAR

// If the status is being forced, use the force value from control,
// else set the control force value to the status
IF inout_stStatus.bForced THEN
	inout_stStatus.bForceValue := inout_stControl.bForceValue;
ELSE
	inout_stControl.bForceValue := inout_stStatus.bForceValue;
END_IF

// Control gets information from the status
inout_stControl.strDevice := inout_stStatus.strDevice;
inout_stControl.strAddress := inout_stStatus.strAddress;
inout_stControl.strLabel := inout_stStatus.strLabel;
inout_stControl.udintLabelId := inout_stStatus.udintLabelId;
inout_stControl.bValue := inout_stStatus.bValue;
inout_stControl.bForced := inout_stStatus.bForced;

END_FUNCTION

// Concrete/IO Mapping/F_SetDigitalIO
(* Links values to a given digital IO struct. *)
FUNCTION F_SetDigitalIO : BOOL
VAR_INPUT
	(* Name of the external device this digital IO is connected to. *)
	in_strDevice: T_MaxString;
	(* Address of this digital IO. *)
	in_strAddress: T_MaxString;
	(* Simple label for this digital IO. *)
	in_strLabel: T_MaxString;
	(* ID of the label for language switching. *)
	in_udintLabelId: UDINT;
	(* Normal input value of this digital IO. *)
	in_bValue: BOOL;
	(* Set to TRUE to force the output. *)
	in_bForce: BOOL;
	(* Must be TRUE to change forced value. *)
	in_bForceInterlock: BOOL;
END_VAR
VAR_IN_OUT
	(* Digital IO struct storing the information about this digital IO. *)
	inout_stIO: ST_DigitalIO;
END_VAR
VAR_OUTPUT
	(* Resulting output value of this digital IO. *)
	out_bValue: BOOL;
END_VAR
VAR
	(* Stores the current value. *)
	bValue: BOOL;
END_VAR

inout_stIO.udintLabelId := in_udintLabelId;
inout_stIO.strDevice := in_strDevice;
inout_stIO.strAddress := in_strAddress;
inout_stIO.strLabel := in_strLabel;
IF in_bForce THEN
	IF in_bForceInterlock THEN
		inout_stIO.bForced := TRUE;
		bValue := inout_stIO.bForceValue;
	ELSE
		inout_stIO.bForced := FALSE;
	END_IF
ELSE
	inout_stIO.bForced := FALSE;
	bValue := in_bValue;
	inout_stIO.bForceValue := bValue;
END_IF
out_bValue := bValue;
inout_stIO.bValue := bValue;

END_FUNCTION

// Concrete/Light Control/FB_PackMLIndicators
FUNCTION_BLOCK FB_PackMLIndicators EXTENDS FB_Module
VAR_INPUT
	(* Machine state. *)
	in_enumState: E_PackMLState;
	(* Machine is suspended due to upstream rather than downstream. *)
	in_bStarvedUpstream: BOOL;
	(* Machine material needs to be refilled. *)
	in_bMaterialShortage: BOOL;
	(* Timing of flashing indicators. *)
	in_timeFlashTiming: TIME := T#250MS;
	(* Time to sound horn for. *)
	in_timeHornTiming: TIME := T#1S;
END_VAR
VAR_OUTPUT
	(* LT red lamp control. *)
	out_bRed: BOOL;
	(* LT yellow lamp control. *)
	out_bYellow: BOOL;
	(* LT blue lamp control. *)
	out_bBlue: BOOL;
	(* LT green lamp control. *)
	out_bGreen: BOOL;
	(* Horn output. *)
	out_bHorn: BOOL;
	(* Start button lamp control. *)
	out_bStartButton: BOOL;
	(* Reset button lamp control. *)
	out_bResetButton: BOOL;
END_VAR
VAR
	fbLTFlashTimer: TON;
	bFlash: BOOL;
	fbHornTimer: TON;
END_VAR

// Flash
fbLTFlashTimer(IN:=TRUE, PT:=in_timeFlashTiming);
IF fbLTFlashTimer.Q THEN
	bFlash := NOT bFlash;
	fbLTFlashTimer(IN:=FALSE);
END_IF

// Light tower
CASE in_enumState OF
	// Flashing red during abnormal stop. 
	E_PackMLState.ABORTING, E_PackMLState.CLEARING, E_PackMLState.ABORTED:
		out_bRed := bFlash;
		out_bYellow := FALSE;
		out_bBlue := in_bMaterialShortage AND bFlash;
		out_bGreen := FALSE;
			
	// Solid red during controlled stop
	E_PackMLState.COMPLETE, E_PackMLState.STOPPED, E_PackMLState.STOPPING, E_PackMLState.RESETTING:
		out_bRed := TRUE;
		out_bYellow := FALSE;
		out_bBlue := in_bMaterialShortage AND bFlash;
		out_bGreen := FALSE;
		
	// Flashing green while ready to start
	E_PackMLState.IDLE:
		out_bRed := FALSE;
		out_bYellow := FALSE;
		out_bBlue := in_bMaterialShortage AND bFlash;
		out_bGreen := bFlash;
		
	// Solid green while running
	E_PackMLState.STARTING, E_PackMLState.EXECUTE, E_PackMLState.COMPLETING, E_PackMLState.UNHOLDING, E_PackMLState.UNSUSPENDING:
		out_bRed := FALSE;
		out_bYellow := FALSE;
		out_bBlue := in_bMaterialShortage AND bFlash;
		out_bGreen := TRUE;
	
	// Solid blue while held
	E_PackMLState.HOLDING, E_PackMLState.HELD:
		out_bRed := FALSE;
		out_bYellow := FALSE;
		out_bBlue := TRUE;
		out_bGreen := FALSE;
		
	E_PackMLState.SUSPENDING, E_PackMLState.SUSPENDED:
		out_bRed := FALSE;
		out_bYellow := (NOT in_bStarvedUpstream) OR (in_bStarvedUpstream AND bFlash);
		out_bBlue := in_bMaterialShortage AND bFlash;
		out_bGreen := TRUE;
END_CASE

// Horn
CASE in_enumState OF
	// Play horn in states transitioning to execute
	E_PackMLState.STARTING, E_PackMLState.UNHOLDING, E_PackMLState.UNSUSPENDING:
		fbHornTimer(IN:=TRUE, PT:=in_timeHornTiming);
		out_bHorn := NOT fbHornTimer.Q;
ELSE // Horn off
	out_bHorn := FALSE;
	fbHornTimer(IN:=FALSE);
END_CASE

// Buttons
CASE in_enumState OF
	// Flash reset button while waiting for press
	E_PackMLState.ABORTED, E_PackMLState.COMPLETE, E_PackMLState.STOPPED:
		out_bResetButton := bFlash;
		out_bStartButton := FALSE;
	
	// Flash start button while waiting for press
	E_PackMLState.IDLE:
		out_bResetButton := FALSE;
		out_bStartButton := bFlash;
	
	// Start button green while running
	E_PackMLState.STARTING, E_PackMLState.EXECUTE, E_PackMLState.COMPLETING, E_PackMLState.UNHOLDING,
			E_PackMLState.SUSPENDING, E_PackMLState.SUSPENDED, E_PackMLState.UNSUSPENDING:
		out_bResetButton := FALSE;
		out_bStartButton := TRUE;
ELSE // Lights off
	out_bResetButton := FALSE;
	out_bStartButton := FALSE;
END_CASE

END_FUNCTION_BLOCK

// Functions/F_ButtonToggle
FUNCTION F_ButtonToggle : BOOL
VAR_INPUT
END_VAR
VAR_IN_OUT
	inout_bButton: BOOL;
	inout_bLastValue: BOOL;
END_VAR

IF inout_bButton THEN
	IF inout_bLastValue THEN
		inout_bButton := FALSE;
		inout_bLastValue := FALSE;
	ELSE
		inout_bLastValue := TRUE;
	END_IF
ELSE
	inout_bLastValue := FALSE;
END_IF

END_FUNCTION

// Functions/F_CalcCycleTime
FUNCTION F_CalcCycleTime : BOOL
VAR_INPUT
	in_timeStartTime: TIME;
END_VAR
VAR_OUTPUT
	out_timeEndTime: TIME;
	out_timeCycleTime: TIME;
END_VAR

out_timeEndTime := TIME();
out_timeCycleTime := out_timeEndTime - in_timeStartTime;
F_CalcCycleTime := TRUE;

END_FUNCTION

// Interfaces/Obsolete/I_ModularAPI
INTERFACE I_ModularAPI

(* Calls a method on the modular API, and returns true once
	the result of the method is received. *)
METHOD M_CallMethod : BOOL
VAR_INPUT
	(* ID of the module the method is being routed to. *)
	strModuleId: T_MaxString;
	
	(* Name of the API method that will be called. *)
	strMethodName: T_MaxString;
	
	(* An array of array of strings representing the name:value pair
		for all of the required method parameters. *)
	arrParameters: T_ApiMethodParameters;
END_VAR
VAR_OUTPUT
	(* Should be TRUE if the method executed without error. *)
	bSuccessful: BOOL;
	
	(* The return value of the method. *)
	strReturnValue: T_MaxString;
	
	(* Name:value pairs for any outputs of the method. *)
	arrOutputValues: T_ApiMethodParameters;
END_VAR
END_METHOD

(* Should return TRUE if there is a method in this interface that
	is executing. *)
PROPERTY P_bApiBusy : BOOL
GET
END_GET
END_PROPERTY

END_INTERFACE

// Project Information/F_GetCompany
// This function has been automatically generated from the project information.
{attribute 'signature_flag' := '1073741824'}
{attribute 'TcGenerated'}
{attribute 'no-analysis'}
FUNCTION F_GetCompany : WSTRING
VAR_INPUT
	
END_VAR

F_GetCompany := "Sensata Technologies";

END_FUNCTION

// Project Information/F_GetTitle
// This function has been automatically generated from the project information.
{attribute 'signature_flag' := '1073741824'}
{attribute 'TcGenerated'}
{attribute 'no-analysis'}
FUNCTION F_GetTitle : WSTRING
VAR_INPUT
	
END_VAR

F_GetTitle := "Sensata_Utilities";

END_FUNCTION

// Project Information/F_GetVersion
// This function has been automatically generated from the project information.
{attribute 'signature_flag' := '1073741824'}
{attribute 'TcGenerated'}
{attribute 'no-analysis'}
FUNCTION F_GetVersion : ST_LibVersion
VAR_INPUT
	
END_VAR

F_GetVersion.iMajor := 0;
F_GetVersion.iMinor := 0;
F_GetVersion.iBuild := 1;
F_GetVersion.iRevision := 0;

END_FUNCTION
